FUNCTION_BLOCK Test_TStreamAdd_Read_PVOID EXTENDS TUnitTestBase
VAR
    Stream : TStream(StreamLength := 2);
    Bob : INT;
END_VAR



Stream.Init(2);

Stream.Add_PVOID(ADR(Bob));
    
Assertion.AssertEquals_UDINT(
    Expected :=8,
    Actual := Stream.Position,
    VariableName := 'Stream.Position');
    
Stream.Seek(0);

Assertion.AssertEquals_PVOID(
    Expected := ADR(Bob),
    Actual := Stream.Read_PVOID(),
    VariableName := 'Stream.Read_PVOID()');
    
Assertion.AssertEquals_UDINT(
    Expected := 8,
    Actual := Stream.Position,
    VariableName := 'Stream.Position');
    
    
TestFinished();

END_FUNCTION_BLOCK

(* stored: Version 1.1.0.1, ProductVersion 3.1.4024.4
   POU Test_TStreamAdd_Read_PVOID: Id {c846e899-74a2-40bf-930c-0def63562594}, SpecialFunc None *)
